Fanuc KAREL source: IO0081.KL

-- PROVISIONAL review KL for V1013-1; original PC SHA256 43f1e49f50a61410fd0a936ffaa9f55b6ed475b8c1126fe2c71a891f903d51ee
-- Incomplete behavior may be omitted. Consult companion uncertainty JSON. Do not deploy.
PROGRAM IO0081
%NOLOCKGROUP
-- UNRESOLVED_LOCAL_POOL 5 cells at code offset 13; source declarations unknown
-- DIRECT_LOCAL_WORD_ACCESS alone does not prove INTEGER, REAL, or BOOLEAN
BEGIN
  -- UNRESOLVED_PC offsets 0-18; opcodes 2B,2C,7B
  -- UNRESOLVED_PC offsets 23-30; opcodes 9D,23
  -- UNRESOLVED_PC offsets 35-49; opcodes 2E,22,9D,33,35
  -- UNRESOLVED_PC offsets 54-61; opcodes 9D,23
  -- UNRESOLVED_PC offsets 66-77; opcodes 2E,23
  -- UNRESOLVED_PC offsets 82-96; opcodes 2E,19,9C,5B,79
  -- UNRESOLVED_PC offsets 101-115; opcodes 21,9D,52,23
  -- UNRESOLVED_PC offsets 125-129; opcodes 7F
  -- UNRESOLVED_PC offsets 134-138; opcodes 27,AA
  -- UNRESOLVED_PC offsets 143-147; opcodes 7F
END IO0081
